FUNCTION_BLOCK GreenMasterAO_Base
VAR_IN_OUT
	AOut: AnalogOutputs;
END_VAR
VAR_INPUT
	F_QN1: LREAL;
	T_GQ1: LREAL;
	F_GQ1: LREAL;
	C_QN1: LREAL;
	H_QN1: LREAL;	
END_VAR
VAR_OUTPUT
END_VAR
VAR
END_VAR

METHOD SetOverrideF_GQ1 : BOOL
VAR_INPUT
	Override: BOOL;
	OverrideValue: LREAL;
	Parameters: REFERENCE TO GreenMasterBaseParameters;
END_VAR
END_METHOD

METHOD SetOverrideF_QN1 : BOOL
VAR_INPUT
	Override: BOOL;
	OverrideValue: LREAL;
	Parameters: REFERENCE TO GreenMasterBaseParameters;
END_VAR
END_METHOD

METHOD SetOverrideH_QN1 : BOOL
VAR_INPUT
	Override: BOOL;
	OverrideValue: LREAL;
	Parameters: REFERENCE TO GreenMasterBaseParameters;
END_VAR
END_METHOD

METHOD SetOverrideT_GQ1 : BOOL
VAR_INPUT
	Override: BOOL;
	OverrideValue: LREAL;
	Parameters: REFERENCE TO GreenMasterBaseParameters;
END_VAR
END_METHOD

END_FUNCTION_BLOCK

(* stored: Version 1.1.0.1, ProductVersion 3.1.4024.6
   POU GreenMasterAO_Base: Id {2680f0d3-3417-4597-9d49-8dca04627f3d}, SpecialFunc None
   Method SetOverrideF_GQ1: Id {1099c3f3-0753-456b-a3a7-f11e02ebc380}
   Method SetOverrideF_QN1: Id {5894b671-2a0c-4309-a421-d0603eabef93}
   Method SetOverrideH_QN1: Id {44d9dd66-2a30-412b-9f34-7a515cc7ca78}
   Method SetOverrideT_GQ1: Id {260aa01c-e2b5-4a84-93ba-bf8109151de5} *)
